// TIA Portal V17 export
// export: Created 2022-07-20T07:01:25.5713776Z, ExportSetting WithDefaults, DisplayName Totally Integrated Automation Portal, DisplayVersion V17, DisplayName TIA Portal Openness, DisplayVersion V17, DisplayName TIA Portal Version Control Interface, DisplayVersion V17, DisplayName SINAMICS Startdrive Advanced, DisplayVersion V17, DisplayName SINAMICS Startdrive G130, G150, S120, S150, SINAMICS MV, S210, DisplayVersion V17, DisplayName SINAMICS Startdrive G110M, G120, G120C, G120D, G120P, G115D, DisplayVersion V17, DisplayName STEP 7 Professional, DisplayVersion V17, DisplayName STEP 7 Safety, DisplayVersion V17, DisplayName WinCC Advanced, DisplayVersion V17
FUNCTION_BLOCK "FB10231_LAM_LexiumDriver10Positions"   // FB10231, LAD
{ S7_Optimized_Access := 'TRUE' }
VERSION : 0.1
// stored: AutoNumber false, IsIECCheckEnabled false, IsRetainMemResEnabled false, MemoryReserve 100, SetENOAutomatically false, UDAEnableTagReadback false
   VAR_INPUT
      RequestEnableMotor : Bool;
      Drive_In : "TLexium_MDrv_Drv2Plc";
      HoldCurrent : SInt;
      RunCurrent : SInt;
      UnitByMotorTurn : LReal := 1.0;
      MicroStepResolution : DInt := 25;   // 256*200 = 51200 microstep/rev max ; Attention, certaines valeur interdites
      RequestAbsolutePositionning : Bool;
      RequestPosition1 : Bool;
      PositionValue1 : Real;
      RequestPosition2 : Bool := false;
      PositionValue2 : Real;
      RequestPosition3 : Bool := false;
      PositionValue3 : Real;
      RequestPosition4 : Bool := false;
      PositionValue4 : Real;
      RequestPosition5 : Bool := false;
      PositionValue5 : Real;
      RequestPosition6 : Bool;
      PositionValue6 : Real;
      RequestPosition7 : Bool;
      PositionValue7 : Real;
      RequestPosition8 : Bool;
      PositionValue8 : Real;
      RequestPosition9 : Bool;
      PositionValue9 : Real;
      RequestPosition10 : Bool;
      PositionValue10 : Real;
      SpeedUnitBySec : Real := 10.0;
      AccelUnitBySec2 : DInt := 100;
      DecelUnitBySec2 : DInt := 100;
      InitialSpeedUnitBySec : DInt := 1;
      RequestHomingInPositiveDirection : Bool;
      RequestJogPositive : Bool;
      RequestJogNegative : Bool;
      JogSpeedUnitBySec : Real;
      HomingSpeedUnitBySec : Real;
      UnitFactor : DInt := 10;
      RequestAcknowledge : Bool;
   END_VAR
   VAR_OUTPUT
      Drive_Out : "TLexium_MDrv_Plc2Drv";
      MotorEnabled : Bool;
      ActualPositionInUnit : Real;
      ActualPositionMicroStep : DInt;
      HomingDone : Bool;
      IsInPosition_1 : Bool;
      IsInPosition_2 : Bool;
      IsInPosition_3 : Bool;
      IsInPosition_4 : Bool;
      IsInPosition_5 : Bool;
      IsInPosition_6 : Bool;
      IsInPosition_7 : Bool;
      IsInPosition_8 : Bool;
      IsInPosition_9 : Bool;
      IsInPosition_10 : Bool;
      Error : Bool;
      ErrorCode : UInt;
   END_VAR
   VAR
      FB10230_LAM_LexiumDriver_Instance { S7_SetPoint := 'True'} : "FB10230_LAM_LexiumDriver";
      MoveType { S7_SetPoint := 'True'} : DInt;
      PosInUnitToMicrostep : DInt;
      SpeedMicrostep : DInt;
      InitialSpeedMicrostep : DInt;
      JogMicrostep : DInt;
      AccelMicroStep2 : DInt;
      DecelMicroStep2 : DInt;
      LocalReqestStartPosition : Bool;
      LocalHomingRequest : Bool;
      LocalHomingMode : SInt := 1;
      RTrig_RequestHoming : R_TRIG;
      HomingInProgress { S7_SetPoint := 'True'} : Bool;
      FTrig_HomingDone : F_TRIG;
      InputsSetup : Array[0..18] of Char;
      temp_uint : UInt;
      i : UInt;
      M_AckEnable : Bool;
      TOF_Enable { S7_SetPoint := 'True'} : TOF_TIME;
      P_HomingDone { S7_SetPoint := 'True'} : Bool;
      LocalUnitByMotorTurn : DInt;
   END_VAR
   // Drive_Out.AS := 2;   // 2 = Mode hybride
   VAR_TEMP   // added for the SCL form of the ladder/FBD networks
      _w1 : Bool;
      _w2 : Bool;
   END_VAR
BEGIN

REGION Network 1 (SCL): Move mode selection
   IF #RequestAbsolutePositionning THEN
       #MoveType := 0;
       #Drive_Out.AS := 2; // Hybride mode
   ELSE
       #MoveType := 1;
   END_IF;
END_REGION

REGION Network 2 (SCL): Unit By Motor Turn Precision
   #LocalUnitByMotorTurn := TRUNC(#UnitByMotorTurn * 100);
END_REGION

REGION Network 3 (SCL): Compute position in microstep
   IF #RequestPosition1 THEN
       #PosInUnitToMicrostep := ((TRUNC(#PositionValue1 * DINT_TO_REAL(#UnitFactor)) * (#MicroStepResolution * 200)) / (#LocalUnitByMotorTurn * #UnitFactor)) * 100;
   ELSIF #RequestPosition2 THEN
       #PosInUnitToMicrostep := ((TRUNC(#PositionValue2 * DINT_TO_REAL(#UnitFactor)) * (#MicroStepResolution * 200)) / (#LocalUnitByMotorTurn * #UnitFactor)) * 100;
   ELSIF #RequestPosition3 THEN
       #PosInUnitToMicrostep := ((TRUNC(#PositionValue3 * DINT_TO_REAL(#UnitFactor)) * (#MicroStepResolution * 200)) / (#LocalUnitByMotorTurn * #UnitFactor)) * 100;
   ELSIF #RequestPosition4 THEN
       #PosInUnitToMicrostep := ((TRUNC(#PositionValue4 * DINT_TO_REAL(#UnitFactor)) * (#MicroStepResolution * 200)) / (#LocalUnitByMotorTurn * #UnitFactor)) * 100;
   ELSIF #RequestPosition5 THEN
       #PosInUnitToMicrostep := ((TRUNC(#PositionValue5 * DINT_TO_REAL(#UnitFactor)) * (#MicroStepResolution * 200)) / (#LocalUnitByMotorTurn * #UnitFactor)) * 100;
   ELSIF #RequestPosition6 THEN
       #PosInUnitToMicrostep := ((TRUNC(#PositionValue6 * DINT_TO_REAL(#UnitFactor)) * (#MicroStepResolution * 200)) / (#LocalUnitByMotorTurn * #UnitFactor)) * 100;
   ELSIF #RequestPosition7 THEN
       #PosInUnitToMicrostep := ((TRUNC(#PositionValue7 * DINT_TO_REAL(#UnitFactor)) * (#MicroStepResolution * 200)) / (#LocalUnitByMotorTurn * #UnitFactor)) * 100;
   ELSIF #RequestPosition8 THEN
       #PosInUnitToMicrostep := ((TRUNC(#PositionValue8 * DINT_TO_REAL(#UnitFactor)) * (#MicroStepResolution * 200)) / (#LocalUnitByMotorTurn * #UnitFactor)) * 100;
   ELSIF #RequestPosition9 THEN
       #PosInUnitToMicrostep := ((TRUNC(#PositionValue9 * DINT_TO_REAL(#UnitFactor)) * (#MicroStepResolution * 200)) / (#LocalUnitByMotorTurn * #UnitFactor)) * 100;
   ELSIF #RequestPosition10 THEN
       #PosInUnitToMicrostep := ((TRUNC(#PositionValue10 * DINT_TO_REAL(#UnitFactor)) * (#MicroStepResolution * 200)) / (#LocalUnitByMotorTurn * #UnitFactor)) * 100;
   END_IF;
END_REGION

REGION Network 4 (SCL): Homing command request
   #RTrig_RequestHoming(CLK := #RequestHomingInPositiveDirection AND (#FB10230_LAM_LexiumDriver_Instance.Drive_In.DE=1) AND (#FB10230_LAM_LexiumDriver_Instance.Drive_In.VM=#SpeedMicrostep));
   #FTrig_HomingDone(CLK := #FB10230_LAM_LexiumDriver_Instance.HM_Act);

   #LocalHomingRequest := #RTrig_RequestHoming.Q AND NOT #FB10230_LAM_LexiumDriver_Instance.ER;

   IF #LocalHomingRequest THEN
       #HomingDone := FALSE;
       #HomingInProgress := TRUE;
   END_IF;

   IF #HomingInProgress AND (#FTrig_HomingDone.Q OR (#FB10230_LAM_LexiumDriver_Instance.ER AND #FB10230_LAM_LexiumDriver_Instance.Error_Code <>85)) THEN
       IF (NOT #FB10230_LAM_LexiumDriver_Instance.ER) OR (#FB10230_LAM_LexiumDriver_Instance.Error_Code = 85) THEN
           #HomingDone := TRUE;

       END_IF;
       #HomingInProgress := FALSE;
   END_IF;

   IF NOT #RequestEnableMotor THEN
       #HomingInProgress := FALSE;
   END_IF;
END_REGION

REGION Network 5 (SCL): Compute speed in microstep
   #SpeedMicrostep := (REAL_TO_DINT((100*#SpeedUnitBySec * DINT_TO_REAL(#MicroStepResolution * 200) / DINT_TO_REAL(#LocalUnitByMotorTurn))));
   IF #SpeedMicrostep >= #MicroStepResolution * 10000 THEN
       #SpeedMicrostep := #MicroStepResolution * 10000;
   END_IF;

   #AccelMicroStep2 := ((#AccelUnitBySec2 * #MicroStepResolution * 200) / #LocalUnitByMotorTurn) * 100;
   IF #AccelMicroStep2 >= #MicroStepResolution *10000 THEN
       #AccelMicroStep2 := #MicroStepResolution *10000;
   END_IF;

   #DecelMicroStep2 := ((#DecelUnitBySec2 * #MicroStepResolution * 200) / #LocalUnitByMotorTurn) * 100;
   IF #DecelMicroStep2 >= #MicroStepResolution *10000 THEN
       #DecelMicroStep2 := #MicroStepResolution *10000;
   END_IF;

   #InitialSpeedMicrostep := 200;//(#InitialSpeedUnitBySec * #MicroStepResolution * 200) / #LocalUnitByMotorTurn;
   IF #InitialSpeedMicrostep >= #SpeedMicrostep THEN
       #InitialSpeedMicrostep := #SpeedMicrostep / 2;
   END_IF;


   IF #HomingInProgress THEN
       #InitialSpeedMicrostep := 200;
       //#SpeedMicrostep := 100;
       (*
       IF #HomingSpeedUnitBySec <> 0 THEN
           #SpeedMicrostep := (REAL_TO_DINT((#HomingSpeedUnitBySec * DINT_TO_REAL(#MicroStepResolution * 200) / DINT_TO_REAL(#LocalUnitByMotorTurn)))) * 100;
       ELSE
           #SpeedMicrostep := #MicroStepResolution * 75;
       END_IF;
       *)
   END_IF;

   #JogMicrostep := (REAL_TO_DINT((#JogSpeedUnitBySec * DINT_TO_REAL(#MicroStepResolution * 200) / DINT_TO_REAL(#LocalUnitByMotorTurn)))) * 100;
   IF #JogMicrostep > 10000 THEN
       #JogMicrostep := 10000;
   END_IF;
END_REGION

REGION Network 6 (SCL): Start Local positionning
   IF #RequestAbsolutePositionning THEN
       #LocalReqestStartPosition :=
       (#RequestPosition1 AND #PositionValue1 <> #ActualPositionInUnit) OR
       (#RequestPosition2 AND #PositionValue2 <> #ActualPositionInUnit) OR
       (#RequestPosition3 AND #PositionValue3 <> #ActualPositionInUnit) OR
       (#RequestPosition4 AND #PositionValue4 <> #ActualPositionInUnit) OR
       (#RequestPosition5 AND #PositionValue5 <> #ActualPositionInUnit) OR
       (#RequestPosition6 AND #PositionValue6 <> #ActualPositionInUnit) OR
       (#RequestPosition7 AND #PositionValue7 <> #ActualPositionInUnit) OR
       (#RequestPosition8 AND #PositionValue8 <> #ActualPositionInUnit) OR
       (#RequestPosition9 AND #PositionValue9 <> #ActualPositionInUnit) OR
       (#RequestPosition10 AND #PositionValue10 <> #ActualPositionInUnit);
   ELSE
       #LocalReqestStartPosition :=
       (#RequestPosition1 AND #PositionValue1 <> 0) OR
       (#RequestPosition2 AND #PositionValue2 <> 0) OR
       (#RequestPosition3 AND #PositionValue3 <> 0) OR
       (#RequestPosition4 AND #PositionValue4 <> 0) OR
       (#RequestPosition5 AND #PositionValue5 <> 0) OR
       (#RequestPosition6 AND #PositionValue6 <> 0) OR
       (#RequestPosition7 AND #PositionValue7 <> 0) OR
       (#RequestPosition8 AND #PositionValue8 <> 0) OR
       (#RequestPosition9 AND #PositionValue9 <> 0) OR
       (#RequestPosition10 AND #PositionValue10 <> 0);
   END_IF;
END_REGION

REGION Network 7: Call Lexium Driver manager
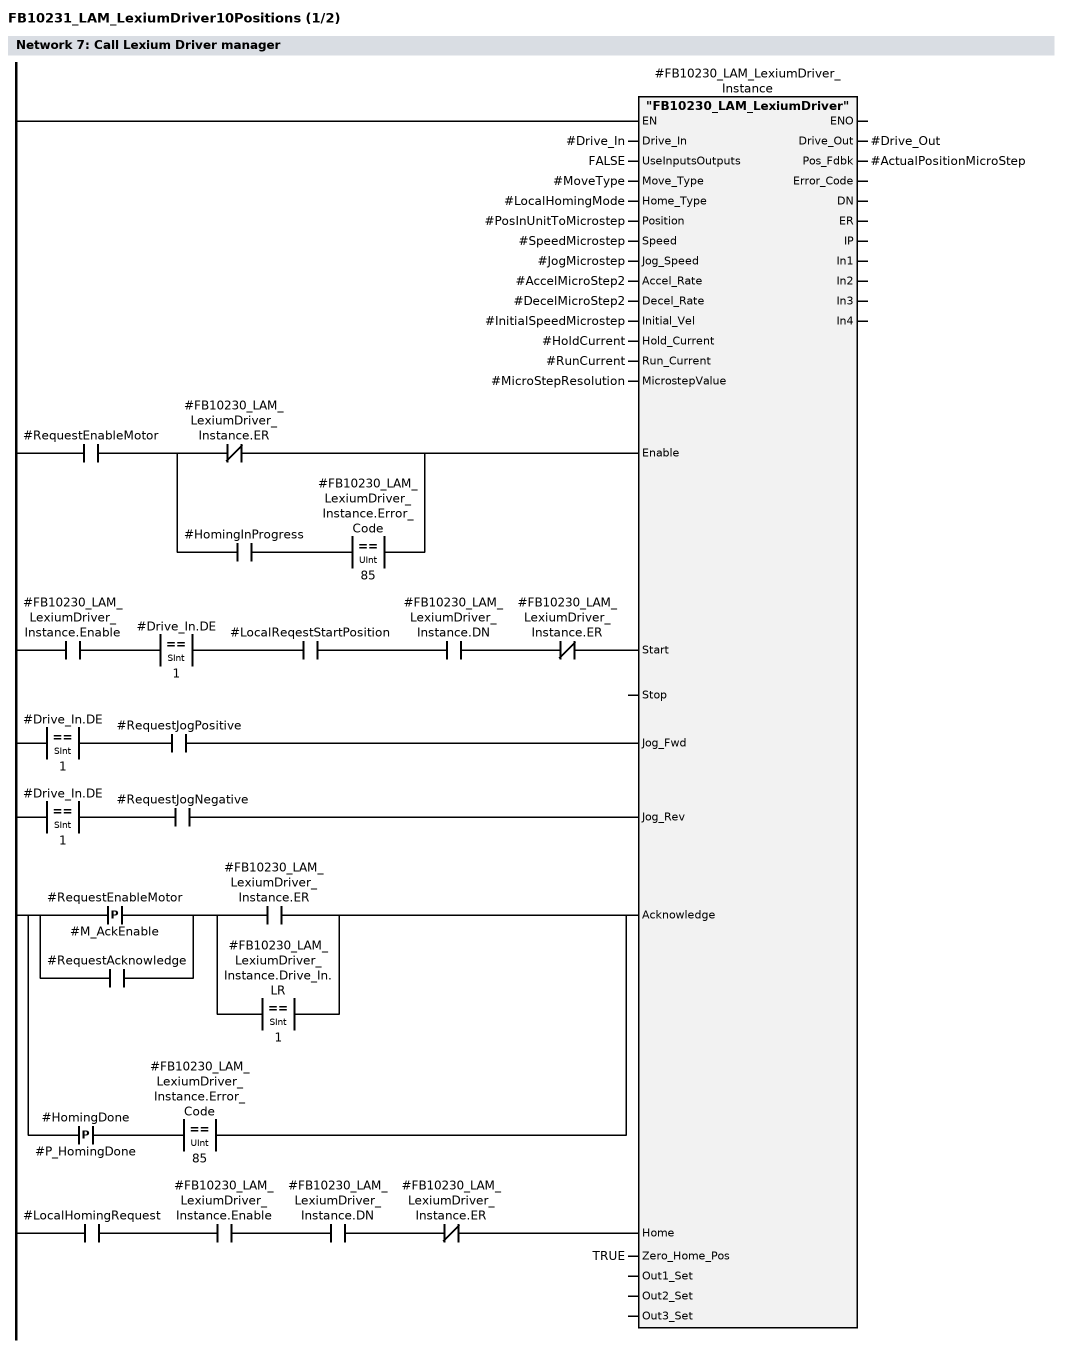
   RUNG wire#powerrail
      #FB10230_LAM_LexiumDriver_Instance(Enable := wire#w2, Start := wire#w3, Jog_Fwd := wire#w4, Jog_Rev := wire#w5, Acknowledge := wire#w7, Home := wire#w8, Drive_In := #Drive_In, UseInputsOutputs := FALSE, Move_Type := #MoveType, Home_Type := #LocalHomingMode, Position := #PosInUnitToMicrostep, Speed := #SpeedMicrostep, Jog_Speed := #JogMicrostep, Accel_Rate := #AccelMicroStep2, Decel_Rate := #DecelMicroStep2, Initial_Vel := #InitialSpeedMicrostep, Hold_Current := #HoldCurrent, Run_Current := #RunCurrent, MicrostepValue := #MicroStepResolution, Stop :=, Zero_Home_Pos := TRUE, Out1_Set :=, Out2_Set :=, Out3_Set :=, Drive_Out => #Drive_Out, Pos_Fdbk => #ActualPositionMicroStep, Error_Code =>, DN =>, ER =>, IP =>, In1 =>, In2 =>, In3 =>, In4 =>)
   END_RUNG
   RUNG wire#powerrail
      Contact( #RequestEnableMotor )
      wire#w1
      I_Contact( #FB10230_LAM_LexiumDriver_Instance.ER )
   END_RUNG wire#w2
   RUNG wire#w1
      Contact( #HomingInProgress )
      { S7_Templates := "SrcType := UInt" } EQ_Contact(in1 := #FB10230_LAM_LexiumDriver_Instance.Error_Code, in2 := 85)
   END_RUNG wire#w2
   RUNG wire#powerrail
      Contact( #FB10230_LAM_LexiumDriver_Instance.Enable )
      { S7_Templates := "SrcType := SInt" } EQ_Contact(in1 := #Drive_In.DE, in2 := 1)
      Contact( #LocalReqestStartPosition )
      Contact( #FB10230_LAM_LexiumDriver_Instance.DN )
      I_Contact( #FB10230_LAM_LexiumDriver_Instance.ER )
   END_RUNG wire#w3
   RUNG wire#powerrail
      { S7_Templates := "SrcType := SInt" } EQ_Contact(in1 := #Drive_In.DE, in2 := 1)
      Contact( #RequestJogPositive )
   END_RUNG wire#w4
   RUNG wire#powerrail
      { S7_Templates := "SrcType := SInt" } EQ_Contact(in1 := #Drive_In.DE, in2 := 1)
      Contact( #RequestJogNegative )
   END_RUNG wire#w5
   RUNG wire#powerrail
      P_Contact(operand := #RequestEnableMotor, bit := #M_AckEnable)
      wire#w6
      Contact( #FB10230_LAM_LexiumDriver_Instance.ER )
   END_RUNG wire#w7
   RUNG wire#powerrail
      Contact( #RequestAcknowledge )
   END_RUNG wire#w6
   RUNG wire#w6
      { S7_Templates := "SrcType := SInt" } EQ_Contact(in1 := #FB10230_LAM_LexiumDriver_Instance.Drive_In.LR, in2 := 1)
   END_RUNG wire#w7
   RUNG wire#powerrail
      P_Contact(operand := #HomingDone, bit := #P_HomingDone)
      { S7_Templates := "SrcType := UInt" } EQ_Contact(in1 := #FB10230_LAM_LexiumDriver_Instance.Error_Code, in2 := 85)
   END_RUNG wire#w7
   RUNG wire#powerrail
      Contact( #LocalHomingRequest )
      Contact( #FB10230_LAM_LexiumDriver_Instance.Enable )
      Contact( #FB10230_LAM_LexiumDriver_Instance.DN )
      I_Contact( #FB10230_LAM_LexiumDriver_Instance.ER )
   END_RUNG wire#w8
   // the same network as SCL:
   #_w1 := #RequestEnableMotor AND NOT #M_AckEnable;   // rising edge of #RequestEnableMotor
   #M_AckEnable := #RequestEnableMotor;
   #_w2 := #HomingDone AND NOT #P_HomingDone;   // rising edge of #HomingDone
   #P_HomingDone := #HomingDone;
   #FB10230_LAM_LexiumDriver_Instance(Drive_In := #Drive_In,   // "FB10230_LAM_LexiumDriver"
                           UseInputsOutputs := FALSE,
                           Move_Type := #MoveType,
                           Home_Type := #LocalHomingMode,
                           Position := #PosInUnitToMicrostep,
                           Speed := #SpeedMicrostep,
                           Jog_Speed := #JogMicrostep,
                           Accel_Rate := #AccelMicroStep2,
                           Decel_Rate := #DecelMicroStep2,
                           Initial_Vel := #InitialSpeedMicrostep,
                           Hold_Current := #HoldCurrent,
                           Run_Current := #RunCurrent,
                           MicrostepValue := #MicroStepResolution,
                           Enable := #RequestEnableMotor AND (NOT #FB10230_LAM_LexiumDriver_Instance.ER OR (#HomingInProgress AND (#FB10230_LAM_LexiumDriver_Instance.Error_Code = 85))),
                           Start := #FB10230_LAM_LexiumDriver_Instance.Enable AND (#Drive_In.DE = 1) AND #LocalReqestStartPosition AND #FB10230_LAM_LexiumDriver_Instance.DN AND NOT #FB10230_LAM_LexiumDriver_Instance.ER,
                           Jog_Fwd := (#Drive_In.DE = 1) AND #RequestJogPositive,
                           Jog_Rev := (#Drive_In.DE = 1) AND #RequestJogNegative,
                           Acknowledge := ((#_w1 OR #RequestAcknowledge) AND (#FB10230_LAM_LexiumDriver_Instance.ER OR (#FB10230_LAM_LexiumDriver_Instance.Drive_In.LR = 1))) OR (#_w2 AND (#FB10230_LAM_LexiumDriver_Instance.Error_Code = 85)),
                           Home := #LocalHomingRequest AND #FB10230_LAM_LexiumDriver_Instance.Enable AND #FB10230_LAM_LexiumDriver_Instance.DN AND NOT #FB10230_LAM_LexiumDriver_Instance.ER,
                           Zero_Home_Pos := TRUE,
                           Drive_Out => #Drive_Out,
                           Pos_Fdbk => #ActualPositionMicroStep);
END_REGION

REGION Network 8: Error handling
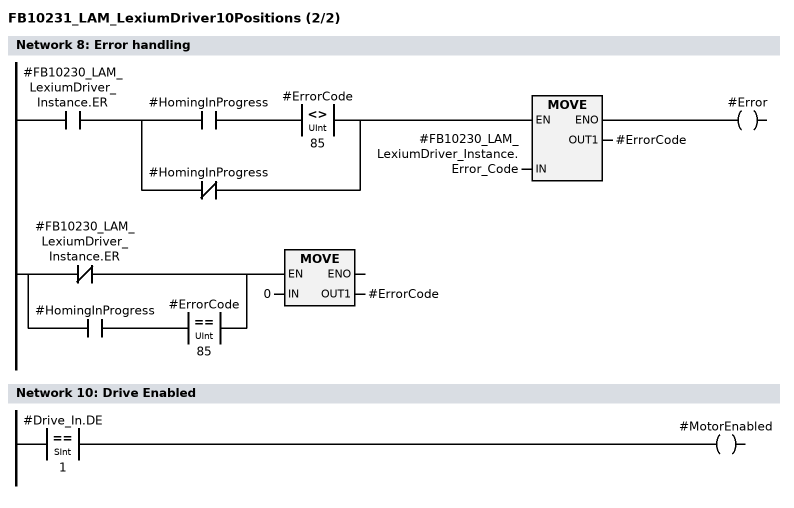
   RUNG wire#powerrail
      Contact( #FB10230_LAM_LexiumDriver_Instance.ER )
      wire#w1
      Contact( #HomingInProgress )
      { S7_Templates := "SrcType := UInt" } NE_Contact(in1 := #ErrorCode, in2 := 85)
      wire#w2
      Move(in := #FB10230_LAM_LexiumDriver_Instance.Error_Code, out1 => #ErrorCode)
      Coil( #Error )
   END_RUNG
   RUNG wire#w1
      I_Contact( #HomingInProgress )
   END_RUNG wire#w2
   RUNG wire#powerrail
      I_Contact( #FB10230_LAM_LexiumDriver_Instance.ER )
      wire#w3
      Move(in := 0, out1 => #ErrorCode)
   END_RUNG
   RUNG wire#powerrail
      Contact( #HomingInProgress )
      { S7_Templates := "SrcType := UInt" } EQ_Contact(in1 := #ErrorCode, in2 := 85)
   END_RUNG wire#w3
   // the same network as SCL:
   #_w1 := #FB10230_LAM_LexiumDriver_Instance.ER AND ((#HomingInProgress AND (#ErrorCode <> 85)) OR NOT #HomingInProgress);
   IF #_w1 THEN #ErrorCode := #FB10230_LAM_LexiumDriver_Instance.Error_Code; END_IF;
   #Error := #_w1;
   IF NOT #FB10230_LAM_LexiumDriver_Instance.ER OR (#HomingInProgress AND (#ErrorCode = 85)) THEN
       #ErrorCode := 0;
   END_IF;
END_REGION

REGION Network 9 (SCL): Actual position in unit
   IF #ActualPositionMicroStep >= 0 THEN
       #ActualPositionInUnit := (DINT_TO_REAL(#ActualPositionMicroStep * #LocalUnitByMotorTurn) / DINT_TO_REAL((#MicroStepResolution * 200)))/100;
   ELSE
       #ActualPositionInUnit := -(((-DINT_TO_REAL(#ActualPositionMicroStep * #LocalUnitByMotorTurn)) / DINT_TO_REAL(#MicroStepResolution * 200)))/100;
   END_IF;
END_REGION

REGION Network 10: Drive Enabled
   RUNG wire#powerrail
      { S7_Templates := "SrcType := SInt" } EQ_Contact(in1 := #Drive_In.DE, in2 := 1)
      Coil( #MotorEnabled )
   END_RUNG
   // the same network as SCL:
   #MotorEnabled := #Drive_In.DE = 1;
END_REGION

REGION Network 11 (SCL): Axis in Position
   //Check Position 1
   #IsInPosition_1 := "FC10021_TolerenceRelation"(X := #PositionValue1, Y := #ActualPositionInUnit, Tolerance := 1.0);

   //Check Position 2
   #IsInPosition_2 := "FC10021_TolerenceRelation"(X := #PositionValue2, Y := #ActualPositionInUnit, Tolerance := 1.0);

   //Check Position 3
   #IsInPosition_3 := "FC10021_TolerenceRelation"(X := #PositionValue3, Y := #ActualPositionInUnit, Tolerance := 1.0);

   //Check Position 4
   #IsInPosition_4 := "FC10021_TolerenceRelation"(X := #PositionValue4, Y := #ActualPositionInUnit, Tolerance := 1.0);

   //Check Position 5
   #IsInPosition_5 := "FC10021_TolerenceRelation"(X := #PositionValue5, Y := #ActualPositionInUnit, Tolerance := 1.0);

   //Check Position 6
   #IsInPosition_6 := "FC10021_TolerenceRelation"(X := #PositionValue3, Y := #ActualPositionInUnit, Tolerance := 1.0);

   //Check Position 7
   #IsInPosition_7 := "FC10021_TolerenceRelation"(X := #PositionValue3, Y := #ActualPositionInUnit, Tolerance := 1.0);

   //Check Position 8
   #IsInPosition_8 := "FC10021_TolerenceRelation"(X := #PositionValue3, Y := #ActualPositionInUnit, Tolerance := 1.0);

   //Check Position 9
   #IsInPosition_9 := "FC10021_TolerenceRelation"(X := #PositionValue3, Y := #ActualPositionInUnit, Tolerance := 1.0);

   //Check Position 10
   #IsInPosition_10 := "FC10021_TolerenceRelation"(X := #PositionValue3, Y := #ActualPositionInUnit, Tolerance := 1.0);
END_REGION
END_FUNCTION_BLOCK
